PROGRAM LON_IN_OUT
VAR
	LON_KL6401: FB_LON_KL6401;
	FB_READ_093_001: FB_READ_093_SNVT_obj_status;
	FB_READ_088_001: FB_READ_088_SNVT_alarm;
	FB_READ_084_001: FB_READ_084_SNVT_time_stamp;
	FB_READ_105_001: FB_READ_105_SNVT_temp_p;
	FB_READ_083_001: FB_READ_083_SNVT_state;
	FB_READ_108_001: FB_READ_108_SNVT_hvac_mode;
	FB_READ_105_002: FB_READ_105_SNVT_temp_p;
	FB_SEND_105_001: FB_SEND_105_SNVT_temp_p;
	F_SNVT_Obj_Status:ARRAY [0..5] OF BYTE;
	F_SNVT_Alarm:ARRAY [0..28] OF BYTE;
	F_SNVT_StateRly:ARRAY [0..1] OF BYTE;

	FB_READ_095_001: FB_READ_095_SNVT_switch;
	F_SNVT_SwitchPwr:ARRAY [0..1] OF BYTE;
	FB_READ_105_003: FB_READ_105_SNVT_temp_p;
	FB_READ_105_004: FB_READ_105_SNVT_temp_p;
	Akt_GB_LON: BOOL;
	FB_SEND_095_001: FB_SEND_095_SNVT_switch;
	F_SNVT_SwitchProdcmd:ARRAY [0..1] OF BYTE;
	FB_SEND_108_001: FB_SEND_108_SNVT_hvac_mode;

	tic						: TON;
	tac						: TON;
	blinker					: BOOL;

	LON_IN_1 	AT %I*:ST_LON_Parameter_IN_36B;
	LON_OUT_1 	AT %Q*:ST_LON_Parameter_OUT_36B;
	stLON_Com_1	: ST_LON_Communication;

	(* Output Variablen *)
	av_GB331_LON_nvo_Node_Status	: INT;
	av_GB331_LON_nvo_Node_Alarm 	: INT;
	av_GB331_LON_nvo_Node_OA_Temp	: REAL;
	av_GB331_LON_nvo_HCC1_Eff_Set	: REAL;
	av_GB331_LON_nvo_Node_RLY_Sta	: INT;
	av_GB331_LON_nvo_HCC1_Unit_St	: INT;
	av_GB331_LON_nviCFDMPwrState_in	: INT;
	av_GB331_LON_nviCFDMSupplyT_in	: REAL;
	av_GB331_LON_nviCFDMEffSetpt_in	: REAL;



	(* Input Variablen *)
	av_GB331_LON_nvi_HCC1_Flow_T	: REAL;
	av_GB331_LON_nvoCFDMProdCmd_out	: REAL;
	av_GB331_LON_nvoCFDMSetpoint_out: REAL;





END_VAR
VAR // added by the converter: edge detectors and wires of the graphical bodies
    _w1 : INT;
    _w2 : ANY;
END_VAR

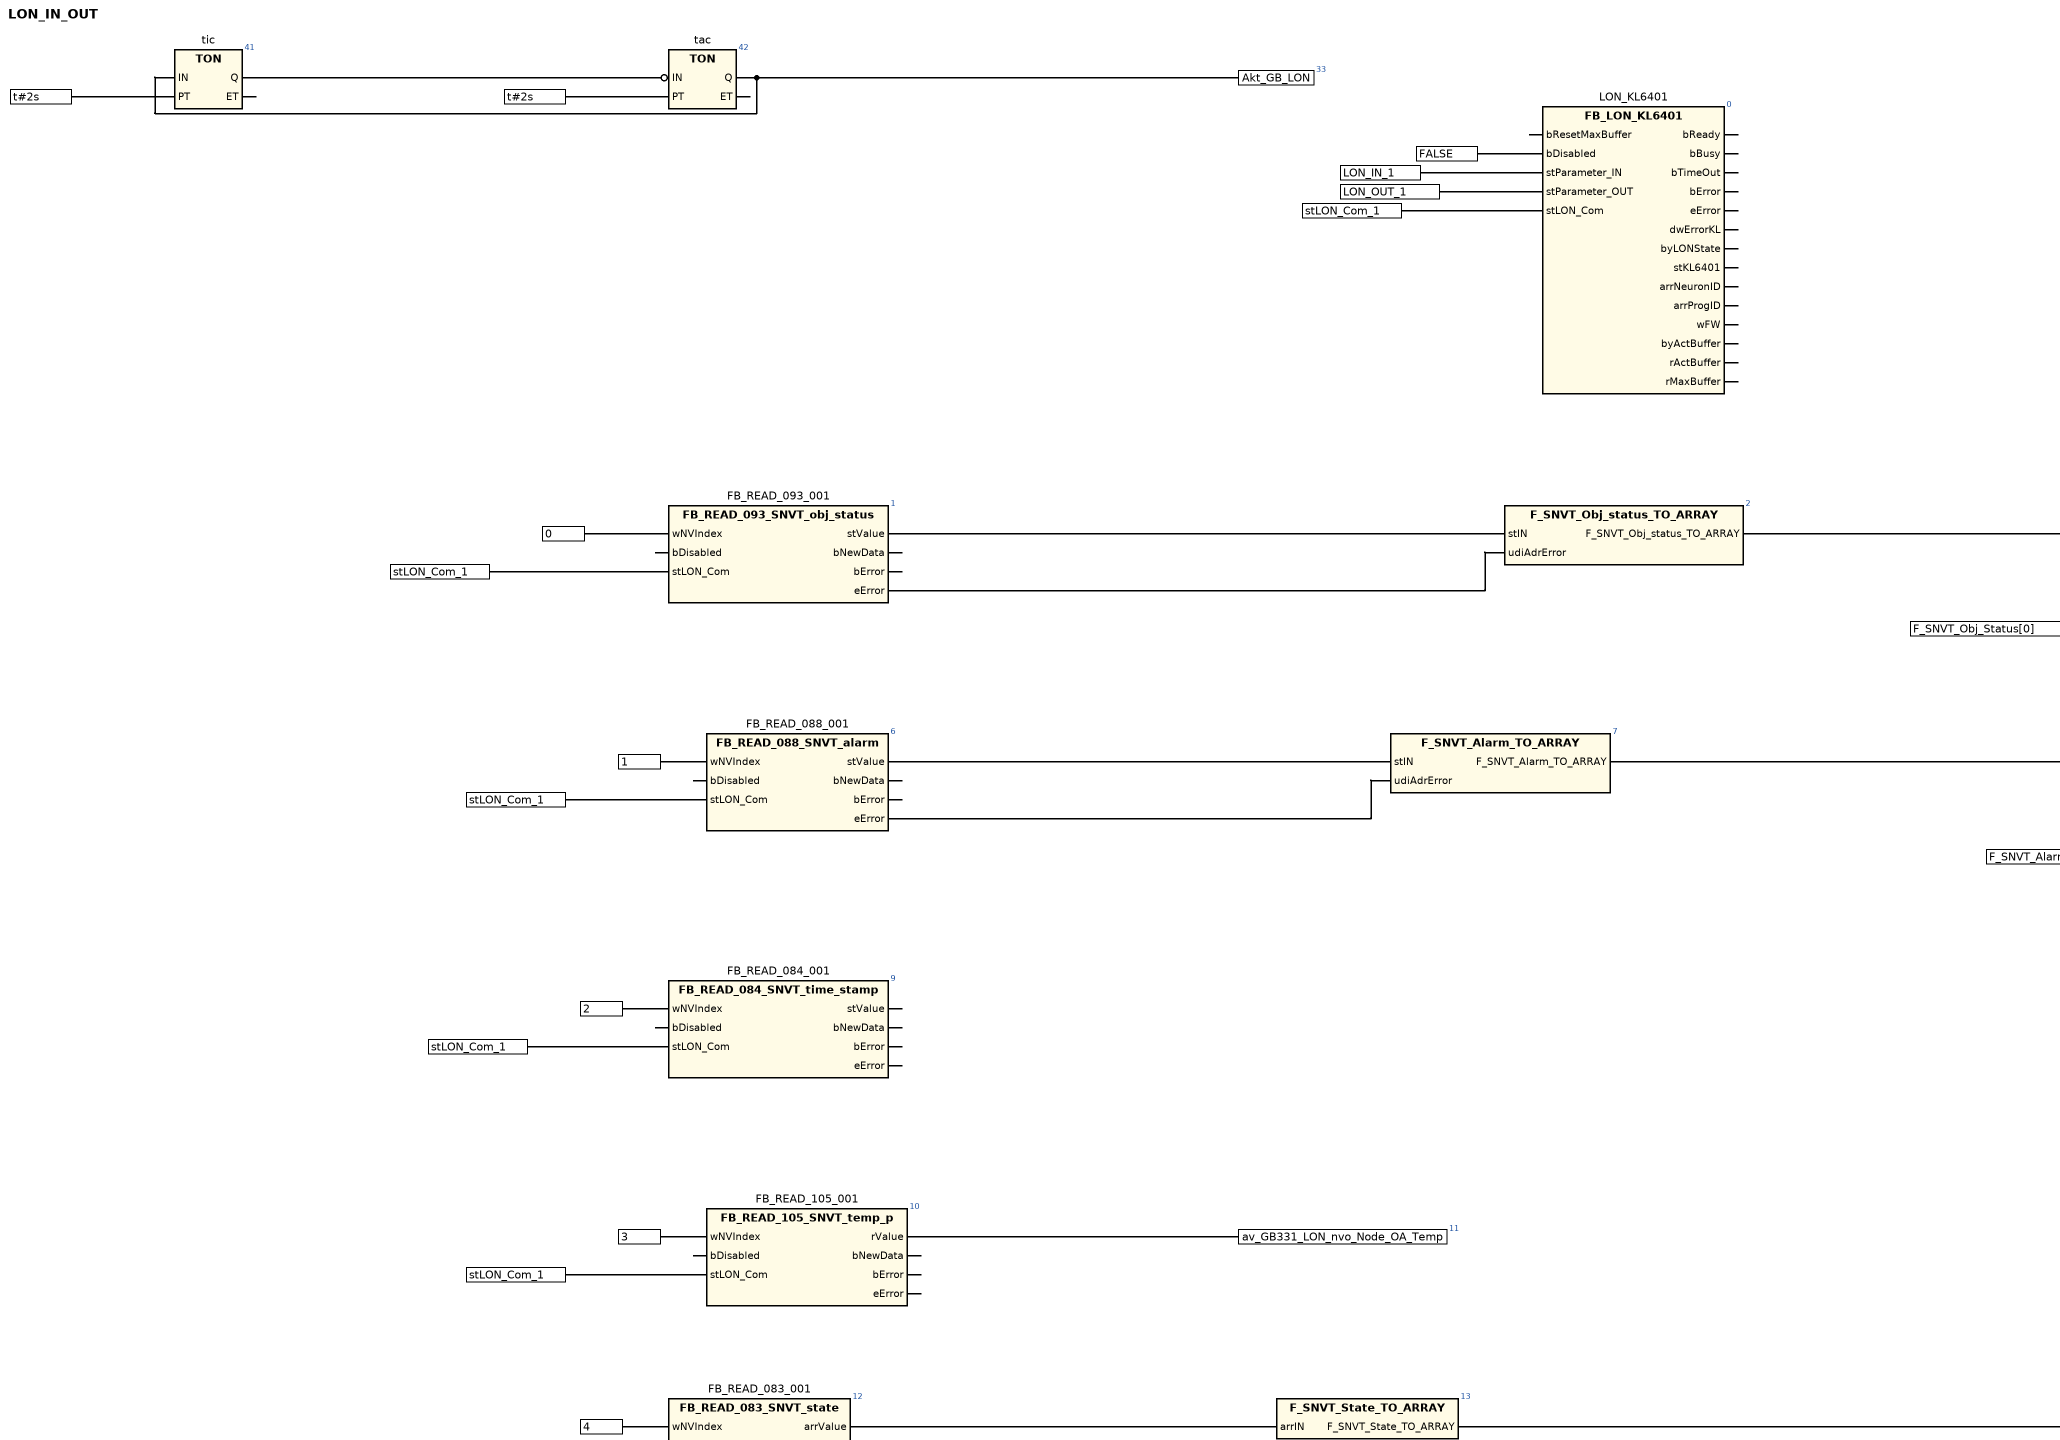
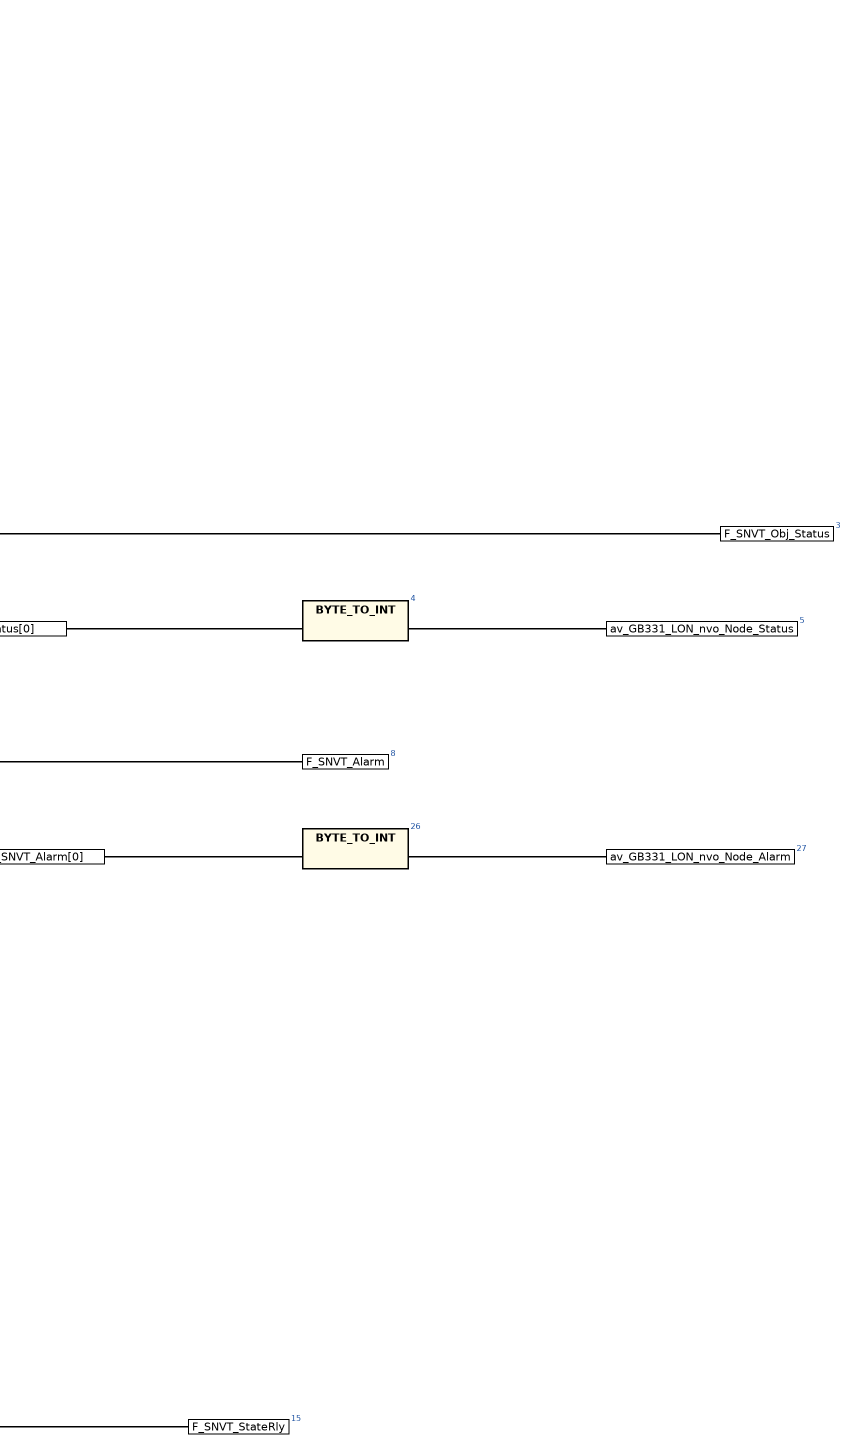
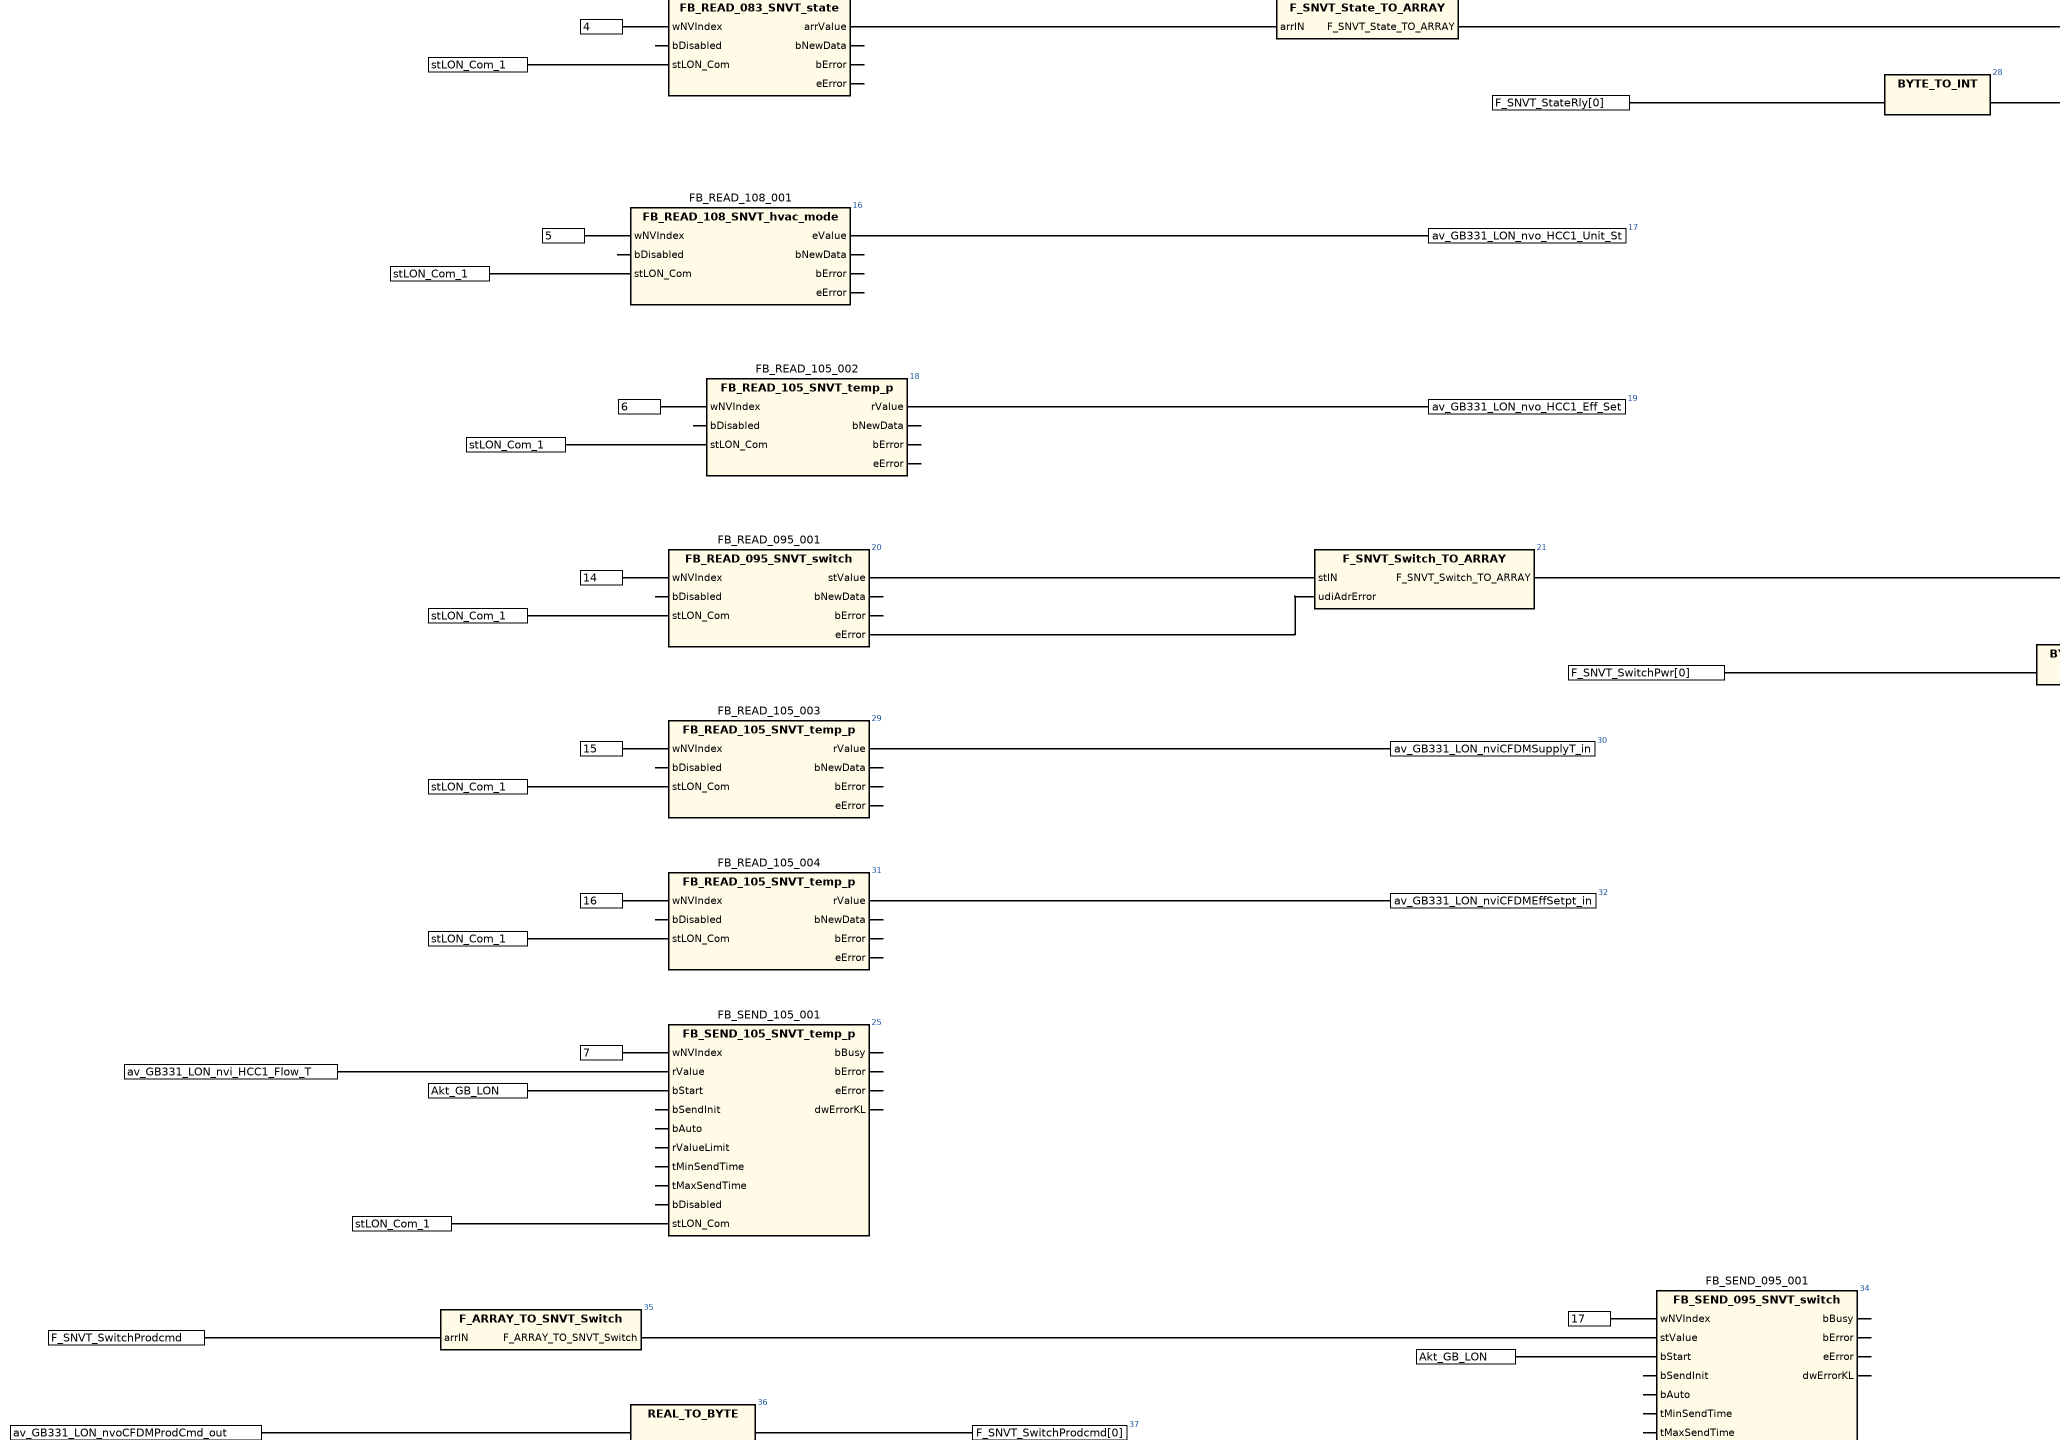
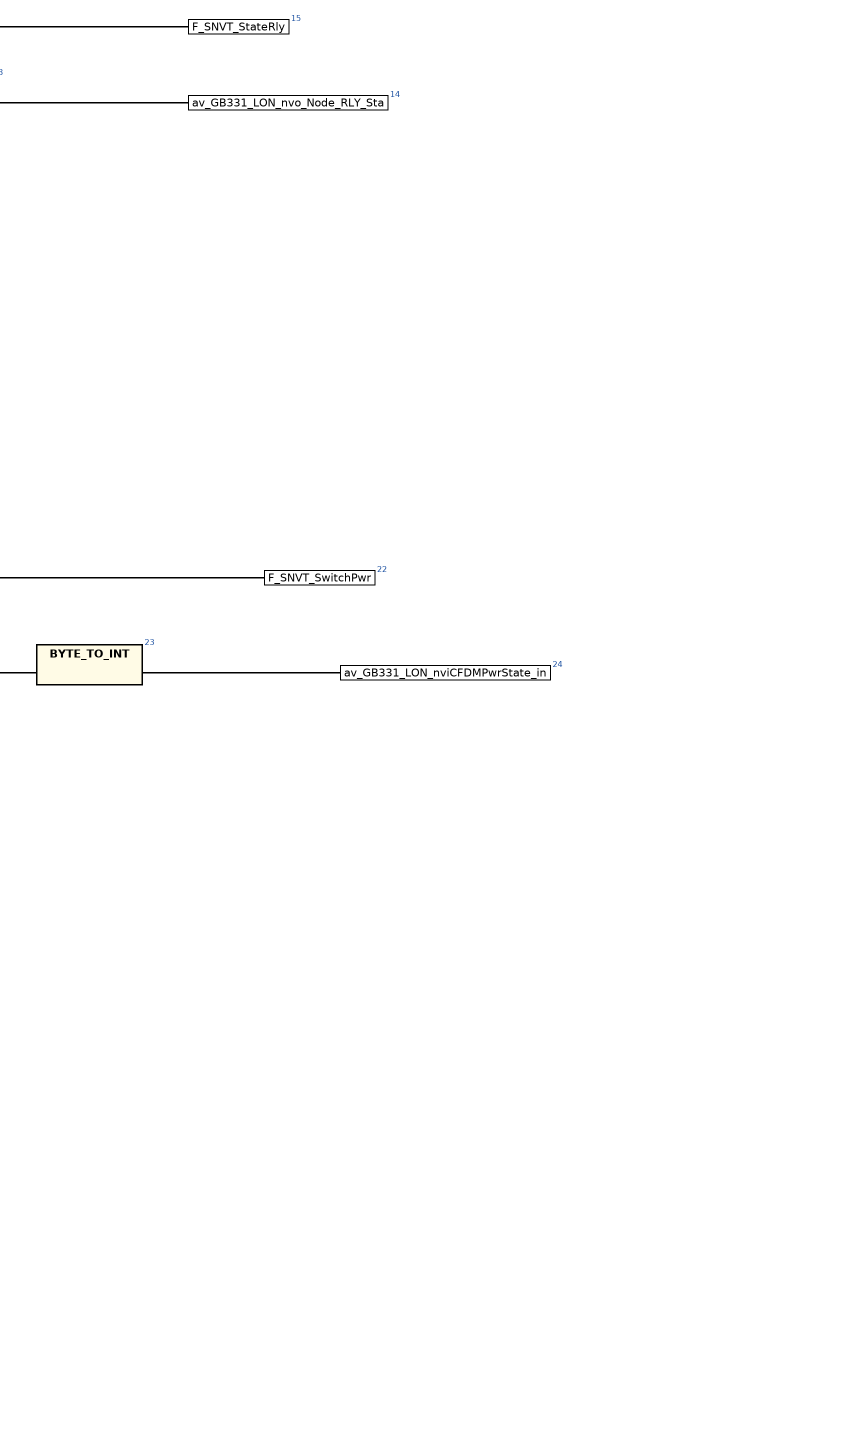
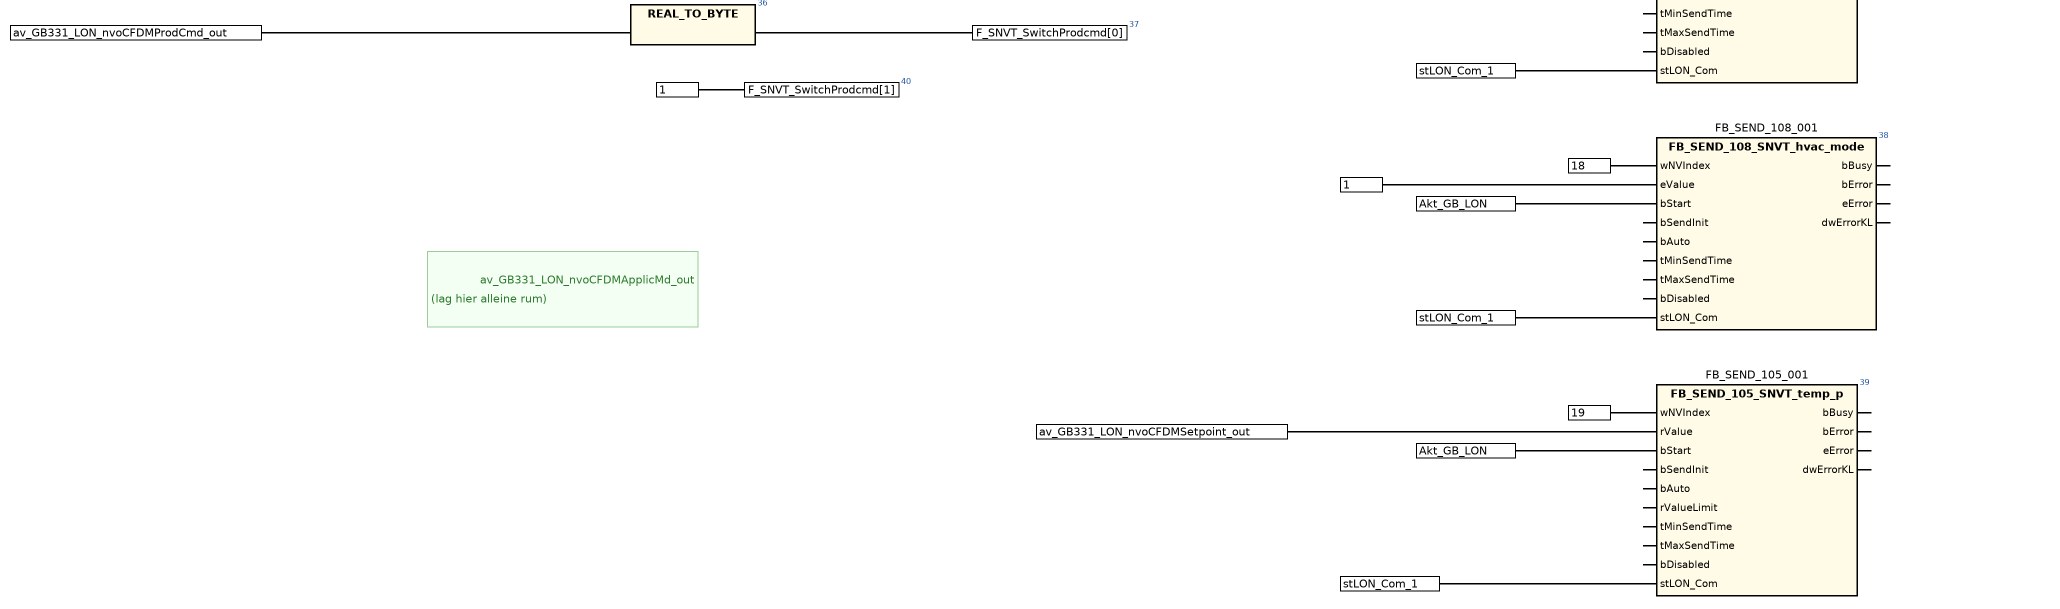
LON_KL6401(
    bDisabled := FALSE,
    stParameter_IN := LON_IN_1,
    stParameter_OUT := LON_OUT_1,
    stLON_Com := stLON_Com_1); // FB_LON_KL6401
FB_READ_093_001(wNVIndex := 0, stLON_Com := stLON_Com_1); // FB_READ_093_SNVT_obj_status
F_SNVT_Obj_Status := F_SNVT_Obj_status_TO_ARRAY(stIN := FB_READ_093_001.stValue, udiAdrError := FB_READ_093_001.eError);
av_GB331_LON_nvo_Node_Status := BYTE_TO_INT(F_SNVT_Obj_Status[0]);
FB_READ_088_001(wNVIndex := 1, stLON_Com := stLON_Com_1); // FB_READ_088_SNVT_alarm
F_SNVT_Alarm := F_SNVT_Alarm_TO_ARRAY(stIN := FB_READ_088_001.stValue, udiAdrError := FB_READ_088_001.eError);
FB_READ_084_001(wNVIndex := 2, stLON_Com := stLON_Com_1); // FB_READ_084_SNVT_time_stamp
FB_READ_105_001(wNVIndex := 3, stLON_Com := stLON_Com_1); // FB_READ_105_SNVT_temp_p
av_GB331_LON_nvo_Node_OA_Temp := FB_READ_105_001.rValue;
FB_READ_083_001(wNVIndex := 4, stLON_Com := stLON_Com_1); // FB_READ_083_SNVT_state
av_GB331_LON_nvo_Node_RLY_Sta := _w1;
F_SNVT_StateRly := F_SNVT_State_TO_ARRAY(arrIN := FB_READ_083_001.arrValue);
FB_READ_108_001(wNVIndex := 5, stLON_Com := stLON_Com_1); // FB_READ_108_SNVT_hvac_mode
av_GB331_LON_nvo_HCC1_Unit_St := FB_READ_108_001.eValue;
FB_READ_105_002(wNVIndex := 6, stLON_Com := stLON_Com_1); // FB_READ_105_SNVT_temp_p
av_GB331_LON_nvo_HCC1_Eff_Set := FB_READ_105_002.rValue;
FB_READ_095_001(wNVIndex := 14, stLON_Com := stLON_Com_1); // FB_READ_095_SNVT_switch
F_SNVT_SwitchPwr := F_SNVT_Switch_TO_ARRAY(stIN := FB_READ_095_001.stValue, udiAdrError := FB_READ_095_001.eError);
av_GB331_LON_nviCFDMPwrState_in := BYTE_TO_INT(F_SNVT_SwitchPwr[0]);
FB_SEND_105_001(
    wNVIndex := 7,
    rValue := av_GB331_LON_nvi_HCC1_Flow_T,
    bStart := Akt_GB_LON,
    stLON_Com := stLON_Com_1); // FB_SEND_105_SNVT_temp_p
av_GB331_LON_nvo_Node_Alarm := BYTE_TO_INT(F_SNVT_Alarm[0]);
_w1 := BYTE_TO_INT(F_SNVT_StateRly[0]);
FB_READ_105_003(wNVIndex := 15, stLON_Com := stLON_Com_1); // FB_READ_105_SNVT_temp_p
av_GB331_LON_nviCFDMSupplyT_in := FB_READ_105_003.rValue;
FB_READ_105_004(wNVIndex := 16, stLON_Com := stLON_Com_1); // FB_READ_105_SNVT_temp_p
av_GB331_LON_nviCFDMEffSetpt_in := FB_READ_105_004.rValue;
Akt_GB_LON := tac.Q;
FB_SEND_095_001(wNVIndex := 17, stValue := _w2, bStart := Akt_GB_LON, stLON_Com := stLON_Com_1); // FB_SEND_095_SNVT_switch
_w2 := F_ARRAY_TO_SNVT_Switch(arrIN := F_SNVT_SwitchProdcmd);
F_SNVT_SwitchProdcmd[0] := REAL_TO_BYTE(av_GB331_LON_nvoCFDMProdCmd_out);
FB_SEND_108_001(wNVIndex := 18, eValue := 1, bStart := Akt_GB_LON, stLON_Com := stLON_Com_1); // FB_SEND_108_SNVT_hvac_mode
FB_SEND_105_001(
    wNVIndex := 19,
    rValue := av_GB331_LON_nvoCFDMSetpoint_out,
    bStart := Akt_GB_LON,
    stLON_Com := stLON_Com_1); // FB_SEND_105_SNVT_temp_p
// 							av_GB331_LON_nvoCFDMApplicMd_out
// (lag hier alleine rum)
//
F_SNVT_SwitchProdcmd[1] := 1;
tic(IN := tac.Q, PT := t#2s); // TON
tac(IN := NOT tic.Q, PT := t#2s); // TON

END_PROGRAM

(* stored: Version 1.1.0.1, ProductVersion 3.1.4024.9
   POU LON_IN_OUT: Id {5b2f3ce2-ae1c-45e1-830a-78c0b64acfcb}, SpecialFunc None *)
